Fanuc KAREL source: ko00038.KL

-- PROVISIONAL review KL for V1013-1; original PC SHA256 950a2199a1d0f779718af7e3fbdac24aeb376ce01ca45a6e326fc08eb05f2563
-- Incomplete behavior may be omitted. Consult companion uncertainty JSON. Do not deploy.
PROGRAM KO00038
%NOLOCKGROUP
BEGIN
  -- UNRESOLVED_PC offsets 5-12; opcodes 9D,23
  -- UNRESOLVED_PC offsets 17-69; opcodes 27,27,49,7E,AD,27,49,7E,AD,22,31,7E,4A
  -- UNRESOLVED_PC offsets 74-78; opcodes 7F
END KO00038
